ABB RobotStudio station: RoboX0_20211201-105547.rsstn

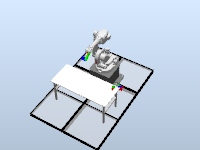
Station RoboX0 (saved by RobotStudio 21.3.9648.0)
Controller IRB1600_10_145, task T_ROB1: task frame (RAPID world) sits at (0, 0, 520) mm in the station
Controller IRB1600_10_145
  mechanical unit ROB_1: IRB1600_10_145__01_2, 6 joints, base frame (0, 0, 0) mm
Layout (positions relative to the parent item):
  - IRB1600_10_145__01_2 [mechanism, from Robots\IRB1600_10_145_G_01.rslib] at (0, 0, 520) mm; joint values [0, 0, 0.0094, 0, 0.5142, 0] (rad or m)
  - подставка [part, from Libraries\box.rslib]
  - Стол сборка_4 [part, from Libraries\table.rslib] at (975, 0, 0) mm, rotated rx 0 ry 0 rz 90 deg
  - gripper2 [mechanism, from Libraries\gripper.rslib] at (806.29, 0, 1668.33) mm, rotated rx -180 ry 60 rz -180 deg; joint values [0] (rad or m)
Attachment: gripper2 is attached to IRB1600_10_145__01_2 / Link6
Targets, tools, work objects and paths stored in the station, written as RAPID:
! task T_ROB1
MODULE CalibData
  TASK PERS wobjdata Workobject_1:=[FALSE,TRUE,"",[[606.263,790,210],[0.707106781,0,0,0.707106781]],[[-100,-100,0],[0,-0.707106781,0.707106781,0]]];
  PERS tooldata gripper:=[TRUE,[[0,0,115],[1,0,0,0]],[0.5,[0,0,30],[1,0,0,0],0,0,0]];
ENDMODULE

! task T_ROB1
MODULE Module1
  CONST robtarget Target_10:=[[199.621572681,690,-886.5],[0,0.5,0,0.866025404],[0,0,0,0],[9E+09,9E+09,9E+09,9E+09,9E+09,9E+09]];
  PROC Path_10()
    MoveL Target_10,v1000,z100,gripper\WObj:=Workobject_1;
  ENDPROC
  PROC main()
  ENDPROC
ENDMODULE

